FUNCTION_BLOCK TestSuiteMock EXTENDS UnitTestSuite IMPLEMENTS ITestSuite
VAR_INPUT
END_VAR
VAR_OUTPUT
END_VAR
VAR
    runTestsCounter: UINT := 0;
END_VAR

METHOD runAllTests
runTestsCounter := runTestsCounter + 1;
END_METHOD

PROPERTY runAllTestsExecuted : BOOL
GET
runAllTestsExecuted := runTestsCounter > 0;
END_GET
END_PROPERTY

END_FUNCTION_BLOCK

(* stored: Version 1.1.0.1, ProductVersion 3.1.4022.12
   POU TestSuiteMock: Id {5bbda9de-22f2-4266-a938-78e140dc1517}, SpecialFunc None
   Method runAllTests: Id {eadccbba-9c8a-464d-a9a3-056873eedb5e}
   Property runAllTestsExecuted: Id {929dff9c-8747-463b-8d7c-fde5ea2bd2fe}
   Get Get: Id {0944b336-5b88-4b5b-b252-286a7367535a} *)
